TYPE AX5000_P_0556 :
STRUCT
	Position_interpolator_type:UINT;
END_STRUCT
END_TYPE

(* stored: Version 1.1.0.1, ProductVersion 3.1.4024.3
   DUT AX5000_P_0556: Id {ab655d63-a17f-4422-8e69-02dbb940bad0} *)
